KUKA KRL data list: Fadenlegen.dat

&ACCESS RVP
&REL 20
&PARAM DISKPATH = KRC:\R1\myProgramme\Mahlen
DEFDAT  Fadenlegen
;FOLD EXTERNAL DECLARATIONS;%{PE}%MKUKATPBASIS,%CEXT,%VCOMMON,%P
;FOLD BASISTECH EXT;%{PE}%MKUKATPBASIS,%CEXT,%VEXT,%P
EXT  BAS (BAS_COMMAND  :IN,REAL  :IN )
;ENDFOLD (BASISTECH EXT)
;FOLD USER EXT;%{E}%MKUKATPUSER,%CEXT,%VEXT,%P
;Make your modifications here

DECL E6POS KM={X 270.508820,Y 129.418152,Z 50.0000,A 0.0,B -180.000,C 0.0,S 6,T 26,E1 0.0,E2 0.0,E3 0.0,E4 0.0,E5 0.0,E6 0.0}

DECL E6POS test1={X 276.364288,Y 142.737,Z 19.5319443,A 180.000,B -180.000,C 0.0,S 2,T 10,E1 0.0,E2 0.0,E3 0.0,E4 0.0,E5 0.0,E6 0.0}

DECL E6AXIS MyHome={A1 13.5221863,A2 -30.7344418,A3 104.022591,A4 -7.46220112,A5 17.3319263,A6 16.0070858,E1 0.0,E2 0.0,E3 0.0,E4 0.0,E5 0.0,E6 0.0}

DECL INT turn=1

DECL INT LetztePos
DECL INT len_Punkte=1435
DECL INT Punkte[1435]

Punkte[1]=113
Punkte[2]=71
Punkte[3]=25
Punkte[4]=159
Punkte[5]=92
Punkte[6]=29
Punkte[7]=161
Punkte[8]=95
Punkte[9]=33
Punkte[10]=84
Punkte[11]=157
Punkte[12]=86
Punkte[13]=128
Punkte[14]=175
Punkte[15]=58
Punkte[16]=9
Punkte[17]=146
Punkte[18]=68
Punkte[19]=113
Punkte[20]=4
Punkte[21]=140
Punkte[22]=5
Punkte[23]=56
Punkte[24]=172
Punkte[25]=119
Punkte[26]=14
Punkte[27]=152
Punkte[28]=80
Punkte[29]=123
Punkte[30]=21
Punkte[31]=156
Punkte[32]=87
Punkte[33]=131
Punkte[34]=177
Punkte[35]=60
Punkte[36]=8
Punkte[37]=144
Punkte[38]=61
Punkte[39]=13
Punkte[40]=150
Punkte[41]=72
Punkte[42]=116
Punkte[43]=9
Punkte[44]=145
Punkte[45]=66
Punkte[46]=112
Punkte[47]=178
Punkte[48]=62
Punkte[49]=110
Punkte[50]=176
Punkte[51]=61
Punkte[52]=143
Punkte[53]=62
Punkte[54]=109
Punkte[55]=172
Punkte[56]=122
Punkte[57]=22
Punkte[58]=158
Punkte[59]=92
Punkte[60]=140
Punkte[61]=3
Punkte[62]=138
Punkte[63]=91
Punkte[64]=35
Punkte[65]=89
Punkte[66]=133
Punkte[67]=179
Punkte[68]=61
Punkte[69]=109
Punkte[70]=173
Punkte[71]=122
Punkte[72]=21
Punkte[73]=157
Punkte[74]=87
Punkte[75]=130
Punkte[76]=177
Punkte[77]=58
Punkte[78]=3
Punkte[79]=139
Punkte[80]=95
Punkte[81]=32
Punkte[82]=163
Punkte[83]=102
Punkte[84]=157
Punkte[85]=91
Punkte[86]=30
Punkte[87]=162
Punkte[88]=97
Punkte[89]=147
Punkte[90]=67
Punkte[91]=23
Punkte[92]=124
Punkte[93]=26
Punkte[94]=159
Punkte[95]=94
Punkte[96]=140
Punkte[97]=2
Punkte[98]=136
Punkte[99]=91
Punkte[100]=163
Punkte[101]=103
Punkte[102]=156
Punkte[103]=88
Punkte[104]=35
Punkte[105]=90
Punkte[106]=157
Punkte[107]=88
Punkte[108]=132
Punkte[109]=179
Punkte[110]=60
Punkte[111]=108
Punkte[112]=168
Punkte[113]=113
Punkte[114]=1
Punkte[115]=136
Punkte[116]=93
Punkte[117]=31
Punkte[118]=163
Punkte[119]=101
Punkte[120]=152
Punkte[121]=76
Punkte[122]=119
Punkte[123]=13
Punkte[124]=151
Punkte[125]=77
Punkte[126]=120
Punkte[127]=16
Punkte[128]=153
Punkte[129]=80
Punkte[130]=122
Punkte[131]=23
Punkte[132]=157
Punkte[133]=89
Punkte[134]=134
Punkte[135]=177
Punkte[136]=57
Punkte[137]=8
Punkte[138]=145
Punkte[139]=64
Punkte[140]=111
Punkte[141]=179
Punkte[142]=134
Punkte[143]=178
Punkte[144]=60
Punkte[145]=107
Punkte[146]=167
Punkte[147]=109
Punkte[148]=170
Punkte[149]=116
Punkte[150]=10
Punkte[151]=147
Punkte[152]=70
Punkte[153]=115
Punkte[154]=6
Punkte[155]=143
Punkte[156]=63
Punkte[157]=110
Punkte[158]=177
Punkte[159]=61
Punkte[160]=108
Punkte[161]=167
Punkte[162]=113
Punkte[163]=0
Punkte[164]=135
Punkte[165]=92
Punkte[166]=31
Punkte[167]=164
Punkte[168]=103
Punkte[169]=159
Punkte[170]=90
Punkte[171]=132
Punkte[172]=177
Punkte[173]=59
Punkte[174]=9
Punkte[175]=147
Punkte[176]=66
Punkte[177]=111
Punkte[178]=177
Punkte[179]=129
Punkte[180]=85
Punkte[181]=128
Punkte[182]=176
Punkte[183]=60
Punkte[184]=106
Punkte[185]=164
Punkte[186]=102
Punkte[187]=153
Punkte[188]=81
Punkte[189]=124
Punkte[190]=24
Punkte[191]=159
Punkte[192]=91
Punkte[193]=29
Punkte[194]=162
Punkte[195]=100
Punkte[196]=153
Punkte[197]=82
Punkte[198]=126
Punkte[199]=28
Punkte[200]=160
Punkte[201]=95
Punkte[202]=142
Punkte[203]=6
Punkte[204]=144
Punkte[205]=64
Punkte[206]=110
Punkte[207]=178
Punkte[208]=131
Punkte[209]=89
Punkte[210]=156
Punkte[211]=85
Punkte[212]=127
Punkte[213]=30
Punkte[214]=161
Punkte[215]=99
Punkte[216]=149
Punkte[217]=70
Punkte[218]=114
Punkte[219]=5
Punkte[220]=141
Punkte[221]=96
Punkte[222]=145
Punkte[223]=63
Punkte[224]=109
Punkte[225]=175
Punkte[226]=59
Punkte[227]=108
Punkte[228]=172
Punkte[229]=124
Punkte[230]=25
Punkte[231]=160
Punkte[232]=97
Punkte[233]=145
Punkte[234]=62
Punkte[235]=108
Punkte[236]=173
Punkte[237]=123
Punkte[238]=25
Punkte[239]=161
Punkte[240]=98
Punkte[241]=146
Punkte[242]=65
Punkte[243]=111
Punkte[244]=176
Punkte[245]=127
Punkte[246]=83
Punkte[247]=126
Punkte[248]=26
Punkte[249]=160
Punkte[250]=96
Punkte[251]=35
Punkte[252]=165
Punkte[253]=109
Punkte[254]=171
Punkte[255]=119
Punkte[256]=16
Punkte[257]=154
Punkte[258]=83
Punkte[259]=125
Punkte[260]=25
Punkte[261]=24
Punkte[262]=158
Punkte[263]=89
Punkte[264]=132
Punkte[265]=178
Punkte[266]=59
Punkte[267]=107
Punkte[268]=166
Punkte[269]=109
Punkte[270]=174
Punkte[271]=123
Punkte[272]=24
Punkte[273]=160
Punkte[274]=92
Punkte[275]=138
Punkte[276]=1
Punkte[277]=57
Punkte[278]=2
Punkte[279]=138
Punkte[280]=93
Punkte[281]=33
Punkte[282]=163
Punkte[283]=100
Punkte[284]=149
Punkte[285]=69
Punkte[286]=114
Punkte[287]=3
Punkte[288]=141
Punkte[289]=93
Punkte[290]=30
Punkte[291]=163
Punkte[292]=50
Punkte[293]=159
Punkte[294]=93
Punkte[295]=32
Punkte[296]=164
Punkte[297]=52
Punkte[298]=168
Punkte[299]=116
Punkte[300]=8
Punkte[301]=146
Punkte[302]=64
Punkte[303]=109
Punkte[304]=41
Punkte[305]=111
Punkte[306]=174
Punkte[307]=124
Punkte[308]=82
Punkte[309]=125
Punkte[310]=26
Punkte[311]=161
Punkte[312]=97
Punkte[313]=143
Punkte[314]=5
Punkte[315]=112
Punkte[316]=2
Punkte[317]=137
Punkte[318]=91
Punkte[319]=158
Punkte[320]=90
Punkte[321]=131
Punkte[322]=176
Punkte[323]=56
Punkte[324]=4
Punkte[325]=139
Punkte[326]=94
Punkte[327]=31
Punkte[328]=165
Punkte[329]=108
Punkte[330]=171
Punkte[331]=123
Punkte[332]=23
Punkte[333]=160
Punkte[334]=49
Punkte[335]=161
Punkte[336]=96
Punkte[337]=144
Punkte[338]=7
Punkte[339]=143
Punkte[340]=95
Punkte[341]=141
Punkte[342]=4
Punkte[343]=142
Punkte[344]=5
Punkte[345]=58
Punkte[346]=176
Punkte[347]=129
Punkte[348]=87
Punkte[349]=132
Punkte[350]=176
Punkte[351]=59
Punkte[352]=106
Punkte[353]=166
Punkte[354]=39
Punkte[355]=105
Punkte[356]=161
Punkte[357]=101
Punkte[358]=154
Punkte[359]=84
Punkte[360]=128
Punkte[361]=174
Punkte[362]=125
Punkte[363]=27
Punkte[364]=160
Punkte[365]=50
Punkte[366]=164
Punkte[367]=35
Punkte[368]=98
Punkte[369]=147
Punkte[370]=65
Punkte[371]=110
Punkte[372]=172
Punkte[373]=125
Punkte[374]=28
Punkte[375]=161
Punkte[376]=50
Punkte[377]=165
Punkte[378]=37
Punkte[379]=102
Punkte[380]=154
Punkte[381]=79
Punkte[382]=121
Punkte[383]=18
Punkte[384]=154
Punkte[385]=81
Punkte[386]=123
Punkte[387]=22
Punkte[388]=159
Punkte[389]=49
Punkte[390]=158
Punkte[391]=93
Punkte[392]=140
Punkte[393]=1
Punkte[394]=55
Punkte[395]=173
Punkte[396]=124
Punkte[397]=83
Punkte[398]=33
Punkte[399]=164
Punkte[400]=92
Punkte[401]=139
Punkte[402]=2
Punkte[403]=113
Punkte[404]=3
Punkte[405]=142
Punkte[406]=94
Punkte[407]=141
Punkte[408]=2
Punkte[409]=114
Punkte[410]=7
Punkte[411]=145
Punkte[412]=65
Punkte[413]=108
Punkte[414]=41
Punkte[415]=112
Punkte[416]=0
Punkte[417]=138
Punkte[418]=94
Punkte[419]=30
Punkte[420]=164
Punkte[421]=51
Punkte[422]=161
Punkte[423]=100
Punkte[424]=150
Punkte[425]=71
Punkte[426]=115
Punkte[427]=7
Punkte[428]=146
Punkte[429]=67
Punkte[430]=18
Punkte[431]=155
Punkte[432]=86
Punkte[433]=126
Punkte[434]=27
Punkte[435]=161
Punkte[436]=103
Punkte[437]=157
Punkte[438]=20
Punkte[439]=155
Punkte[440]=85
Punkte[441]=125
Punkte[442]=173
Punkte[443]=57
Punkte[444]=107
Punkte[445]=168
Punkte[446]=115
Punkte[447]=8
Punkte[448]=147
Punkte[449]=68
Punkte[450]=112
Punkte[451]=1
Punkte[452]=137
Punkte[453]=92
Punkte[454]=30
Punkte[455]=29
Punkte[456]=126
Punkte[457]=174
Punkte[458]=58
Punkte[459]=107
Punkte[460]=170
Punkte[461]=119
Punkte[462]=75
Punkte[463]=118
Punkte[464]=14
Punkte[465]=153
Punkte[466]=79
Punkte[467]=120
Punkte[468]=19
Punkte[469]=154
Punkte[470]=82
Punkte[471]=123
Punkte[472]=172
Punkte[473]=50
Punkte[474]=158
Punkte[475]=88
Punkte[476]=131
Punkte[477]=130
Punkte[478]=89
Punkte[479]=90
Punkte[480]=135
Punkte[481]=178
Punkte[482]=58
Punkte[483]=106
Punkte[484]=168
Punkte[485]=43
Punkte[486]=100
Punkte[487]=151
Punkte[488]=76
Punkte[489]=118
Punkte[490]=15
Punkte[491]=152
Punkte[492]=77
Punkte[493]=119
Punkte[494]=17
Punkte[495]=153
Punkte[496]=76
Punkte[497]=117
Punkte[498]=9
Punkte[499]=148
Punkte[500]=67
Punkte[501]=113
Punkte[502]=179
Punkte[503]=136
Punkte[504]=92
Punkte[505]=32
Punkte[506]=165
Punkte[507]=103
Punkte[508]=49
Punkte[509]=162
Punkte[510]=101
Punkte[511]=153
Punkte[512]=18
Punkte[513]=156
Punkte[514]=86
Punkte[515]=127
Punkte[516]=28
Punkte[517]=162
Punkte[518]=98
Punkte[519]=145
Punkte[520]=6
Punkte[521]=116
Punkte[522]=11
Punkte[523]=149
Punkte[524]=71
Punkte[525]=114
Punkte[526]=9
Punkte[527]=149
Punkte[528]=73
Punkte[529]=116
Punkte[530]=7
Punkte[531]=147
Punkte[532]=69
Punkte[533]=113
Punkte[534]=5
Punkte[535]=144
Punkte[536]=63
Punkte[537]=108
Punkte[538]=40
Punkte[539]=110
Punkte[540]=175
Punkte[541]=54
Punkte[542]=177
Punkte[543]=62
Punkte[544]=107
Punkte[545]=165
Punkte[546]=36
Punkte[547]=101
Punkte[548]=151
Punkte[549]=14
Punkte[550]=154
Punkte[551]=78
Punkte[552]=121
Punkte[553]=19
Punkte[554]=155
Punkte[555]=83
Punkte[556]=122
Punkte[557]=19
Punkte[558]=156
Punkte[559]=49
Punkte[560]=171
Punkte[561]=121
Punkte[562]=20
Punkte[563]=156
Punkte[564]=100
Punkte[565]=44
Punkte[566]=170
Punkte[567]=118
Punkte[568]=12
Punkte[569]=150
Punkte[570]=75
Punkte[571]=117
Punkte[572]=12
Punkte[573]=151
Punkte[574]=74
Punkte[575]=117
Punkte[576]=8
Punkte[577]=148
Punkte[578]=68
Punkte[579]=111
Punkte[580]=40
Punkte[581]=109
Punkte[582]=66
Punkte[583]=146
Punkte[584]=63
Punkte[585]=107
Punkte[586]=40
Punkte[587]=112
Punkte[588]=177
Punkte[589]=133
Punkte[590]=178
Punkte[591]=61
Punkte[592]=107
Punkte[593]=39
Punkte[594]=102
Punkte[595]=155
Punkte[596]=81
Punkte[597]=122
Punkte[598]=20
Punkte[599]=158
Punkte[600]=83
Punkte[601]=123
Punkte[602]=124
Punkte[603]=27
Punkte[604]=162
Punkte[605]=99
Punkte[606]=147
Punkte[607]=11
Punkte[608]=148
Punkte[609]=70
Punkte[610]=113
Punkte[611]=169
Punkte[612]=117
Punkte[613]=11
Punkte[614]=150
Punkte[615]=98
Punkte[616]=39
Punkte[617]=106
Punkte[618]=55
Punkte[619]=172
Punkte[620]=49
Punkte[621]=102
Punkte[622]=156
Punkte[623]=84
Punkte[624]=127
Punkte[625]=175
Punkte[626]=55
Punkte[627]=170
Punkte[628]=120
Punkte[629]=15
Punkte[630]=153
Punkte[631]=78
Punkte[632]=120
Punkte[633]=20
Punkte[634]=21
Punkte[635]=159
Punkte[636]=85
Punkte[637]=126
Punkte[638]=175
Punkte[639]=56
Punkte[640]=106
Punkte[641]=167
Punkte[642]=114
Punkte[643]=4
Punkte[644]=143
Punkte[645]=94
Punkte[646]=33
Punkte[647]=165
Punkte[648]=52
Punkte[649]=166
Punkte[650]=38
Punkte[651]=102
Punkte[652]=47
Punkte[653]=171
Punkte[654]=122
Punkte[655]=79
Punkte[656]=155
Punkte[657]=87
Punkte[658]=127
Punkte[659]=174
Punkte[660]=55
Punkte[661]=105
Punkte[662]=162
Punkte[663]=102
Punkte[664]=48
Punkte[665]=171
Punkte[666]=118
Punkte[667]=13
Punkte[668]=149
Punkte[669]=72
Punkte[670]=115
Punkte[671]=4
Punkte[672]=144
Punkte[673]=95
Punkte[674]=140
Punkte[675]=139
Punkte[676]=1
Punkte[677]=114
Punkte[678]=42
Punkte[679]=112
Punkte[680]=179
Punkte[681]=178
Punkte[682]=111
Punkte[683]=167
Punkte[684]=41
Punkte[685]=110
Punkte[686]=173
Punkte[687]=121
Punkte[688]=21
Punkte[689]=20
Punkte[690]=19
Punkte[691]=157
Punkte[692]=82
Punkte[693]=121
Punkte[694]=17
Punkte[695]=154
Punkte[696]=80
Punkte[697]=121
Punkte[698]=172
Punkte[699]=48
Punkte[700]=100
Punkte[701]=152
Punkte[702]=75
Punkte[703]=116
Punkte[704]=13
Punkte[705]=152
Punkte[706]=79
Punkte[707]=119
Punkte[708]=15
Punkte[709]=154
Punkte[710]=100
Punkte[711]=45
Punkte[712]=170
Punkte[713]=117
Punkte[714]=10
Punkte[715]=148
Punkte[716]=69
Punkte[717]=111
Punkte[718]=166
Punkte[719]=37
Punkte[720]=101
Punkte[721]=45
Punkte[722]=169
Punkte[723]=114
Punkte[724]=6
Punkte[725]=146
Punkte[726]=96
Punkte[727]=142
Punkte[728]=143
Punkte[729]=96
Punkte[730]=147
Punkte[731]=146
Punkte[732]=10
Punkte[733]=149
Punkte[734]=97
Punkte[735]=144
Punkte[736]=145
Punkte[737]=5
Punkte[738]=115
Punkte[739]=9
Punkte[740]=10
Punkte[741]=150
Punkte[742]=99
Punkte[743]=148
Punkte[744]=71
Punkte[745]=112
Punkte[746]=167
Punkte[747]=40
Punkte[748]=106
Punkte[749]=57
Punkte[750]=174
Punkte[751]=129
Punkte[752]=88
Punkte[753]=34
Punkte[754]=84
Punkte[755]=126
Punkte[756]=173
Punkte[757]=54
Punkte[758]=174
Punkte[759]=53
Punkte[760]=172
Punkte[761]=51
Punkte[762]=165
Punkte[763]=34
Punkte[764]=98
Punkte[765]=40
Punkte[766]=168
Punkte[767]=114
Punkte[768]=72
Punkte[769]=24
Punkte[770]=161
Punkte[771]=104
Punkte[772]=160
Punkte[773]=94
Punkte[774]=137
Punkte[775]=93
Punkte[776]=29
Punkte[777]=163
Punkte[778]=51
Punkte[779]=168
Punkte[780]=42
Punkte[781]=98
Punkte[782]=148
Punkte[783]=72
Punkte[784]=113
Punkte[785]=114
Punkte[786]=41
Punkte[787]=107
Punkte[788]=169
Punkte[789]=116
Punkte[790]=74
Punkte[791]=118
Punkte[792]=10
Punkte[793]=11
Punkte[794]=151
Punkte[795]=98
Punkte[796]=41
Punkte[797]=168
Punkte[798]=112
Punkte[799]=70
Punkte[800]=71
Punkte[801]=72
Punkte[802]=73
Punkte[803]=115
Punkte[804]=169
Punkte[805]=118
Punkte[806]=11
Punkte[807]=12
Punkte[808]=148
Punkte[809]=97
Punkte[810]=146
Punkte[811]=145
Punkte[812]=95
Punkte[813]=36
Punkte[814]=94
Punkte[815]=32
Punkte[816]=33
Punkte[817]=97
Punkte[818]=36
Punkte[819]=166
Punkte[820]=110
Punkte[821]=174
Punkte[822]=51
Punkte[823]=162
Punkte[824]=103
Punkte[825]=50
Punkte[826]=166
Punkte[827]=34
Punkte[828]=97
Punkte[829]=42
Punkte[830]=169
Punkte[831]=54
Punkte[832]=176
Punkte[833]=130
Punkte[834]=86
Punkte[835]=129
Punkte[836]=175
Punkte[837]=57
Punkte[838]=104
Punkte[839]=163
Punkte[840]=99
Punkte[841]=41
Punkte[842]=169
Punkte[843]=53
Punkte[844]=171
Punkte[845]=50
Punkte[846]=162
Punkte[847]=31
Punkte[848]=32
Punkte[849]=33
Punkte[850]=166
Punkte[851]=108
Punkte[852]=169
Punkte[853]=119
Punkte[854]=78
Punkte[855]=152
Punkte[856]=16
Punkte[857]=155
Punkte[858]=84
Punkte[859]=125
Punkte[860]=175
Punkte[861]=53
Punkte[862]=105
Punkte[863]=165
Punkte[864]=164
Punkte[865]=34
Punkte[866]=96
Punkte[867]=33
Punkte[868]=34
Punkte[869]=95
Punkte[870]=166
Punkte[871]=35
Punkte[872]=97
Punkte[873]=41
Punkte[874]=42
Punkte[875]=170
Punkte[876]=115
Punkte[877]=75
Punkte[878]=74
Punkte[879]=26
Punkte[880]=162
Punkte[881]=104
Punkte[882]=159
Punkte[883]=95
Punkte[884]=35
Punkte[885]=167
Punkte[886]=110
Punkte[887]=66
Punkte[888]=67
Punkte[889]=110
Punkte[890]=3
Punkte[891]=2
Punkte[892]=1
Punkte[893]=0
Punkte[894]=111
Punkte[895]=168
Punkte[896]=39
Punkte[897]=104
Punkte[898]=52
Punkte[899]=169
Punkte[900]=43
Punkte[901]=99
Punkte[902]=151
Punkte[903]=15
Punkte[904]=14
Punkte[905]=13
Punkte[906]=153
Punkte[907]=77
Punkte[908]=118
Punkte[909]=17
Punkte[910]=155
Punkte[911]=82
Punkte[912]=122
Punkte[913]=121
Punkte[914]=81
Punkte[915]=125
Punkte[916]=124
Punkte[917]=84
Punkte[918]=83
Punkte[919]=82
Punkte[920]=81
Punkte[921]=120
Punkte[922]=171
Punkte[923]=46
Punkte[924]=170
Punkte[925]=53
Punkte[926]=104
Punkte[927]=164
Punkte[928]=163
Punkte[929]=28
Punkte[930]=76
Punkte[931]=116
Punkte[932]=117
Punkte[933]=13
Punkte[934]=12
Punkte[935]=152
Punkte[936]=99
Punkte[937]=42
Punkte[938]=43
Punkte[939]=170
Punkte[940]=52
Punkte[941]=167
Punkte[942]=39
Punkte[943]=103
Punkte[944]=51
Punkte[945]=169
Punkte[946]=46
Punkte[947]=100
Punkte[948]=38
Punkte[949]=104
Punkte[950]=55
Punkte[951]=176
Punkte[952]=57
Punkte[953]=105
Punkte[954]=160
Punkte[955]=98
Punkte[956]=43
Punkte[957]=44
Punkte[958]=169
Punkte[959]=96
Punkte[960]=37
Punkte[961]=103
Punkte[962]=53
Punkte[963]=167
Punkte[964]=38
Punkte[965]=103
Punkte[966]=52
Punkte[967]=173
Punkte[968]=49
Punkte[969]=100
Punkte[970]=170
Punkte[971]=48
Punkte[972]=101
Punkte[973]=155
Punkte[974]=156
Punkte[975]=17
Punkte[976]=64
Punkte[977]=108
Punkte[978]=39
Punkte[979]=101
Punkte[980]=46
Punkte[981]=172
Punkte[982]=120
Punkte[983]=18
Punkte[984]=19
Punkte[985]=65
Punkte[986]=109
Punkte[987]=39
Punkte[988]=96
Punkte[989]=159
Punkte[990]=102
Punkte[991]=50
Punkte[992]=173
Punkte[993]=56
Punkte[994]=105
Punkte[995]=163
Punkte[996]=162
Punkte[997]=161
Punkte[998]=160
Punkte[999]=93
Punkte[1000]=139
Punkte[1001]=138
Punkte[1002]=137
Punkte[1003]=136
Punkte[1004]=135
Punkte[1005]=134
Punkte[1006]=91
Punkte[1007]=90
Punkte[1008]=89
Punkte[1009]=88
Punkte[1010]=130
Punkte[1011]=175
Punkte[1012]=102
Punkte[1013]=51
Punkte[1014]=166
Punkte[1015]=167
Punkte[1016]=37
Punkte[1017]=98
Punkte[1018]=44
Punkte[1019]=171
Punkte[1020]=117
Punkte[1021]=73
Punkte[1022]=114
Punkte[1023]=115
Punkte[1024]=74
Punkte[1025]=75
Punkte[1026]=76
Punkte[1027]=77
Punkte[1028]=117
Punkte[1029]=118
Punkte[1030]=78
Punkte[1031]=79
Punkte[1032]=80
Punkte[1033]=120
Punkte[1034]=121
Punkte[1035]=122
Punkte[1036]=123
Punkte[1037]=124
Punkte[1038]=125
Punkte[1039]=126
Punkte[1040]=127
Punkte[1041]=128
Punkte[1042]=87
Punkte[1043]=34
Punkte[1044]=94
Punkte[1045]=158
Punkte[1046]=102
Punkte[1047]=52
Punkte[1048]=53
Punkte[1049]=168
Punkte[1050]=38
Punkte[1051]=101
Punkte[1052]=47
Punkte[1053]=170
Punkte[1054]=108
Punkte[1055]=107
Punkte[1056]=106
Punkte[1057]=169
Punkte[1058]=40
Punkte[1059]=104
Punkte[1060]=54
Punkte[1061]=171
Punkte[1062]=45
Punkte[1063]=99
Punkte[1064]=153
Punkte[1065]=154
Punkte[1066]=155
Punkte[1067]=156
Punkte[1068]=101
Punkte[1069]=49
Punkte[1070]=50
Punkte[1071]=101
Punkte[1072]=157
Punkte[1073]=158
Punkte[1074]=103
Punkte[1075]=54
Punkte[1076]=172
Punkte[1077]=47
Punkte[1078]=99
Punkte[1079]=36
Punkte[1080]=167
Punkte[1081]=51
Punkte[1082]=101
Punkte[1083]=102
Punkte[1084]=172
Punkte[1085]=173
Punkte[1086]=174
Punkte[1087]=56
Punkte[1088]=104
Punkte[1089]=105
Punkte[1090]=54
Punkte[1091]=55
Punkte[1092]=103
Punkte[1093]=160
Punkte[1094]=161
Punkte[1095]=162
Punkte[1096]=163
Punkte[1097]=164
Punkte[1098]=165
Punkte[1099]=166
Punkte[1100]=167
Punkte[1101]=97
Punkte[1102]=38
Punkte[1103]=105
Punkte[1104]=58
Punkte[1105]=59
Punkte[1106]=105
Punkte[1107]=40
Punkte[1108]=39
Punkte[1109]=38
Punkte[1110]=37
Punkte[1111]=95
Punkte[1112]=94
Punkte[1113]=35
Punkte[1114]=36
Punkte[1115]=96
Punkte[1116]=97
Punkte[1117]=98
Punkte[1118]=149
Punkte[1119]=12
Punkte[1120]=13
Punkte[1121]=14
Punkte[1122]=15
Punkte[1123]=16
Punkte[1124]=17
Punkte[1125]=18
Punkte[1126]=19
Punkte[1127]=20
Punkte[1128]=21
Punkte[1129]=22
Punkte[1130]=23
Punkte[1131]=24
Punkte[1132]=25
Punkte[1133]=26
Punkte[1134]=27
Punkte[1135]=28
Punkte[1136]=29
Punkte[1137]=30
Punkte[1138]=31
Punkte[1139]=32
Punkte[1140]=33
Punkte[1141]=34
Punkte[1142]=35
Punkte[1143]=36
Punkte[1144]=37
Punkte[1145]=38
Punkte[1146]=39
Punkte[1147]=40
Punkte[1148]=41
Punkte[1149]=42
Punkte[1150]=43
Punkte[1151]=44
Punkte[1152]=99
Punkte[1153]=169
Punkte[1154]=168
Punkte[1155]=99
Punkte[1156]=46
Punkte[1157]=47
Punkte[1158]=100
Punkte[1159]=101
Punkte[1160]=102
Punkte[1161]=53
Punkte[1162]=54
Punkte[1163]=55
Punkte[1164]=56
Punkte[1165]=57
Punkte[1166]=58
Punkte[1167]=59
Punkte[1168]=60
Punkte[1169]=61
Punkte[1170]=106
Punkte[1171]=107
Punkte[1172]=108
Punkte[1173]=109
Punkte[1174]=110
Punkte[1175]=111
Punkte[1176]=175
Punkte[1177]=174
Punkte[1178]=173
Punkte[1179]=172
Punkte[1180]=171
Punkte[1181]=170
Punkte[1182]=169
Punkte[1183]=168
Punkte[1184]=167
Punkte[1185]=166
Punkte[1186]=165
Punkte[1187]=164
Punkte[1188]=163
Punkte[1189]=162
Punkte[1190]=161
Punkte[1191]=160
Punkte[1192]=159
Punkte[1193]=158
Punkte[1194]=157
Punkte[1195]=156
Punkte[1196]=155
Punkte[1197]=154
Punkte[1198]=153
Punkte[1199]=152
Punkte[1200]=151
Punkte[1201]=150
Punkte[1202]=149
Punkte[1203]=148
Punkte[1204]=147
Punkte[1205]=146
Punkte[1206]=145
Punkte[1207]=144
Punkte[1208]=143
Punkte[1209]=142
Punkte[1210]=141
Punkte[1211]=140
Punkte[1212]=139
Punkte[1213]=138
Punkte[1214]=137
Punkte[1215]=136
Punkte[1216]=135
Punkte[1217]=134
Punkte[1218]=133
Punkte[1219]=132
Punkte[1220]=131
Punkte[1221]=130
Punkte[1222]=129
Punkte[1223]=128
Punkte[1224]=127
Punkte[1225]=126
Punkte[1226]=125
Punkte[1227]=124
Punkte[1228]=123
Punkte[1229]=122
Punkte[1230]=121
Punkte[1231]=120
Punkte[1232]=119
Punkte[1233]=118
Punkte[1234]=117
Punkte[1235]=116
Punkte[1236]=115
Punkte[1237]=114
Punkte[1238]=113
Punkte[1239]=112
Punkte[1240]=111
Punkte[1241]=110
Punkte[1242]=109
Punkte[1243]=108
Punkte[1244]=107
Punkte[1245]=106
Punkte[1246]=105
Punkte[1247]=104
Punkte[1248]=103
Punkte[1249]=102
Punkte[1250]=101
Punkte[1251]=100
Punkte[1252]=99
Punkte[1253]=98
Punkte[1254]=45
Punkte[1255]=46
Punkte[1256]=47
Punkte[1257]=48
Punkte[1258]=49
Punkte[1259]=50
Punkte[1260]=51
Punkte[1261]=52
Punkte[1262]=53
Punkte[1263]=54
Punkte[1264]=55
Punkte[1265]=56
Punkte[1266]=57
Punkte[1267]=58
Punkte[1268]=59
Punkte[1269]=60
Punkte[1270]=61
Punkte[1271]=62
Punkte[1272]=63
Punkte[1273]=64
Punkte[1274]=65
Punkte[1275]=66
Punkte[1276]=67
Punkte[1277]=68
Punkte[1278]=69
Punkte[1279]=70
Punkte[1280]=71
Punkte[1281]=72
Punkte[1282]=73
Punkte[1283]=74
Punkte[1284]=75
Punkte[1285]=76
Punkte[1286]=77
Punkte[1287]=78
Punkte[1288]=79
Punkte[1289]=80
Punkte[1290]=81
Punkte[1291]=82
Punkte[1292]=83
Punkte[1293]=84
Punkte[1294]=85
Punkte[1295]=86
Punkte[1296]=87
Punkte[1297]=88
Punkte[1298]=89
Punkte[1299]=90
Punkte[1300]=91
Punkte[1301]=92
Punkte[1302]=93
Punkte[1303]=94
Punkte[1304]=95
Punkte[1305]=96
Punkte[1306]=97
Punkte[1307]=98
Punkte[1308]=99
Punkte[1309]=100
Punkte[1310]=101
Punkte[1311]=102
Punkte[1312]=103
Punkte[1313]=104
Punkte[1314]=105
Punkte[1315]=106
Punkte[1316]=107
Punkte[1317]=108
Punkte[1318]=109
Punkte[1319]=110
Punkte[1320]=111
Punkte[1321]=112
Punkte[1322]=113
Punkte[1323]=114
Punkte[1324]=115
Punkte[1325]=116
Punkte[1326]=117
Punkte[1327]=118
Punkte[1328]=119
Punkte[1329]=120
Punkte[1330]=121
Punkte[1331]=122
Punkte[1332]=123
Punkte[1333]=124
Punkte[1334]=125
Punkte[1335]=126
Punkte[1336]=127
Punkte[1337]=128
Punkte[1338]=129
Punkte[1339]=130
Punkte[1340]=131
Punkte[1341]=132
Punkte[1342]=133
Punkte[1343]=134
Punkte[1344]=135
Punkte[1345]=136
Punkte[1346]=137
Punkte[1347]=138
Punkte[1348]=139
Punkte[1349]=140
Punkte[1350]=141
Punkte[1351]=142
Punkte[1352]=143
Punkte[1353]=144
Punkte[1354]=145
Punkte[1355]=146
Punkte[1356]=147
Punkte[1357]=148
Punkte[1358]=149
Punkte[1359]=150
Punkte[1360]=151
Punkte[1361]=152
Punkte[1362]=153
Punkte[1363]=154
Punkte[1364]=155
Punkte[1365]=156
Punkte[1366]=157
Punkte[1367]=158
Punkte[1368]=159
Punkte[1369]=160
Punkte[1370]=161
Punkte[1371]=162
Punkte[1372]=163
Punkte[1373]=164
Punkte[1374]=165
Punkte[1375]=166
Punkte[1376]=167
Punkte[1377]=168
Punkte[1378]=169
Punkte[1379]=170
Punkte[1380]=171
Punkte[1381]=172
Punkte[1382]=173
Punkte[1383]=174
Punkte[1384]=175
Punkte[1385]=176
Punkte[1386]=177
Punkte[1387]=178
Punkte[1388]=179
Punkte[1389]=180
Punkte[1390]=181
Punkte[1391]=182
Punkte[1392]=183
Punkte[1393]=184
Punkte[1394]=185
Punkte[1395]=186
Punkte[1396]=187
Punkte[1397]=188
Punkte[1398]=189
Punkte[1399]=190
Punkte[1400]=191
Punkte[1401]=192
Punkte[1402]=193
Punkte[1403]=194
Punkte[1404]=195
Punkte[1405]=196
Punkte[1406]=197
Punkte[1407]=198
Punkte[1408]=199
Punkte[1409]=200
Punkte[1410]=201
Punkte[1411]=202
Punkte[1412]=203
Punkte[1413]=204
Punkte[1414]=205
Punkte[1415]=206
Punkte[1416]=207
Punkte[1417]=208
Punkte[1418]=209
Punkte[1419]=210
Punkte[1420]=211
Punkte[1421]=212
Punkte[1422]=213
Punkte[1423]=214
Punkte[1424]=215
Punkte[1425]=216
Punkte[1426]=217
Punkte[1427]=218
Punkte[1428]=219
Punkte[1429]=220
Punkte[1430]=221
Punkte[1431]=222
Punkte[1432]=223
Punkte[1433]=224
Punkte[1434]=225
Punkte[1435]=226


;ENDFOLD (USER EXT)
;ENDFOLD (EXTERNAL DECLARATIONS)
ENDDAT
